// TIA Portal V18 export
DATA_BLOCK "ST10_Flow26_JMagnetLoad&Unload_iDB"   // DB1096
VERSION : 0.1
// stored: AutoNumber false, DBAccessibleFromOPCUA true, DBAccessibleFromWebserver true, InstanceOfName ST10_Flow26_JMagnetLoad&Unload, InstanceOfType FB
"ST10_Flow26_JMagnetLoad&Unload"
   // // inherited from GRAPH_BASE
   // VAR
   //    OFF_SQ_BASE : Bool;
   // END_VAR
   // VAR_INPUT
   //    iSysInface : "RCS_SysComInterface_V1";
   // END_VAR
   // VAR_IN_OUT
   //    ioPM_Inface : "RCS_PMInterface_V1";
   //    ioStatus : Int;
   // END_VAR
   // VAR
   //    sCtrlMode { S7_SetPoint := 'True'} : "SysFlowCtrlGraph";
   //    sUpdMES_Data : Bool;
   //    工件放行中 : Bool;
   //    前站站号 { ExternalAccessible := 'False'; ExternalVisible := 'False'; ExternalWritable := 'False'} : UInt;
   //    本站站号 { ExternalAccessible := 'False'; ExternalVisible := 'False'; ExternalWritable := 'False'} : UInt;
   //    弹窗Temp : Array[1..10] of Int;
   //    AlarmID : Int;
   //    TON { S7_SetPoint := 'True'} : Array[0..10] of TON_TIME;
   //    TOF { S7_SetPoint := 'True'} : Array[0..10] of TOF_TIME;
   //    sUP { S7_SetPoint := 'True'} : Array[0..10] of Bool;
   //    更新RFID完成 : Bool;
   //    RT_DATA { ExternalAccessible := 'False'; ExternalVisible := 'False'; ExternalWritable := 'False'; S7_SetPoint := 'True'} : G7_RTDataPlus_V6;
   //    Trans1 { ExternalAccessible := 'False'; ExternalVisible := 'False'; ExternalWritable := 'False'; S7_SetPoint := 'True'} : G7_TransitionPlus_V6;
   //    Trans2 { ExternalAccessible := 'False'; ExternalVisible := 'False'; ExternalWritable := 'False'; S7_SetPoint := 'True'} : G7_TransitionPlus_V6;
   //    Trans3 { ExternalAccessible := 'False'; ExternalVisible := 'False'; ExternalWritable := 'False'; S7_SetPoint := 'True'} : G7_TransitionPlus_V6;
   //    Trans102 { ExternalAccessible := 'False'; ExternalVisible := 'False'; ExternalWritable := 'False'; S7_SetPoint := 'True'} : G7_TransitionPlus_V6;
   //    Trans28 { ExternalAccessible := 'False'; ExternalVisible := 'False'; ExternalWritable := 'False'; S7_SetPoint := 'True'} : G7_TransitionPlus_V6;
   //    Trans29 { ExternalAccessible := 'False'; ExternalVisible := 'False'; ExternalWritable := 'False'; S7_SetPoint := 'True'} : G7_TransitionPlus_V6;
   //    Trans30 { ExternalAccessible := 'False'; ExternalVisible := 'False'; ExternalWritable := 'False'; S7_SetPoint := 'True'} : G7_TransitionPlus_V6;
   //    Trans31 { ExternalAccessible := 'False'; ExternalVisible := 'False'; ExternalWritable := 'False'; S7_SetPoint := 'True'} : G7_TransitionPlus_V6;
   //    Trans32 { ExternalAccessible := 'False'; ExternalVisible := 'False'; ExternalWritable := 'False'; S7_SetPoint := 'True'} : G7_TransitionPlus_V6;
   //    Trans33 { ExternalAccessible := 'False'; ExternalVisible := 'False'; ExternalWritable := 'False'; S7_SetPoint := 'True'} : G7_TransitionPlus_V6;
   //    Trans34 { ExternalAccessible := 'False'; ExternalVisible := 'False'; ExternalWritable := 'False'; S7_SetPoint := 'True'} : G7_TransitionPlus_V6;
   //    Trans35 { ExternalAccessible := 'False'; ExternalVisible := 'False'; ExternalWritable := 'False'; S7_SetPoint := 'True'} : G7_TransitionPlus_V6;
   //    Trans36 { ExternalAccessible := 'False'; ExternalVisible := 'False'; ExternalWritable := 'False'; S7_SetPoint := 'True'} : G7_TransitionPlus_V6;
   //    Trans37 { ExternalAccessible := 'False'; ExternalVisible := 'False'; ExternalWritable := 'False'; S7_SetPoint := 'True'} : G7_TransitionPlus_V6;
   //    Trans38 { ExternalAccessible := 'False'; ExternalVisible := 'False'; ExternalWritable := 'False'; S7_SetPoint := 'True'} : G7_TransitionPlus_V6;
   //    Trans39 { ExternalAccessible := 'False'; ExternalVisible := 'False'; ExternalWritable := 'False'; S7_SetPoint := 'True'} : G7_TransitionPlus_V6;
   //    Trans40 { ExternalAccessible := 'False'; ExternalVisible := 'False'; ExternalWritable := 'False'; S7_SetPoint := 'True'} : G7_TransitionPlus_V6;
   //    Trans41 { ExternalAccessible := 'False'; ExternalVisible := 'False'; ExternalWritable := 'False'; S7_SetPoint := 'True'} : G7_TransitionPlus_V6;
   //    Trans42 { ExternalAccessible := 'False'; ExternalVisible := 'False'; ExternalWritable := 'False'; S7_SetPoint := 'True'} : G7_TransitionPlus_V6;
   //    Trans43 { ExternalAccessible := 'False'; ExternalVisible := 'False'; ExternalWritable := 'False'; S7_SetPoint := 'True'} : G7_TransitionPlus_V6;
   //    Trans44 { ExternalAccessible := 'False'; ExternalVisible := 'False'; ExternalWritable := 'False'; S7_SetPoint := 'True'} : G7_TransitionPlus_V6;
   //    Trans45 { ExternalAccessible := 'False'; ExternalVisible := 'False'; ExternalWritable := 'False'; S7_SetPoint := 'True'} : G7_TransitionPlus_V6;
   //    Trans46 { ExternalAccessible := 'False'; ExternalVisible := 'False'; ExternalWritable := 'False'; S7_SetPoint := 'True'} : G7_TransitionPlus_V6;
   //    Trans47 { ExternalAccessible := 'False'; ExternalVisible := 'False'; ExternalWritable := 'False'; S7_SetPoint := 'True'} : G7_TransitionPlus_V6;
   //    Trans48 { ExternalAccessible := 'False'; ExternalVisible := 'False'; ExternalWritable := 'False'; S7_SetPoint := 'True'} : G7_TransitionPlus_V6;
   //    Trans49 { ExternalAccessible := 'False'; ExternalVisible := 'False'; ExternalWritable := 'False'; S7_SetPoint := 'True'} : G7_TransitionPlus_V6;
   //    Trans50 { ExternalAccessible := 'False'; ExternalVisible := 'False'; ExternalWritable := 'False'; S7_SetPoint := 'True'} : G7_TransitionPlus_V6;
   //    Trans51 { ExternalAccessible := 'False'; ExternalVisible := 'False'; ExternalWritable := 'False'; S7_SetPoint := 'True'} : G7_TransitionPlus_V6;
   //    Trans52 { ExternalAccessible := 'False'; ExternalVisible := 'False'; ExternalWritable := 'False'; S7_SetPoint := 'True'} : G7_TransitionPlus_V6;
   //    Trans53 { ExternalAccessible := 'False'; ExternalVisible := 'False'; ExternalWritable := 'False'; S7_SetPoint := 'True'} : G7_TransitionPlus_V6;
   //    Trans54 { ExternalAccessible := 'False'; ExternalVisible := 'False'; ExternalWritable := 'False'; S7_SetPoint := 'True'} : G7_TransitionPlus_V6;
   //    Trans55 { ExternalAccessible := 'False'; ExternalVisible := 'False'; ExternalWritable := 'False'; S7_SetPoint := 'True'} : G7_TransitionPlus_V6;
   //    Trans56 { ExternalAccessible := 'False'; ExternalVisible := 'False'; ExternalWritable := 'False'; S7_SetPoint := 'True'} : G7_TransitionPlus_V6;
   //    Trans57 { ExternalAccessible := 'False'; ExternalVisible := 'False'; ExternalWritable := 'False'; S7_SetPoint := 'True'} : G7_TransitionPlus_V6;
   //    Trans58 { ExternalAccessible := 'False'; ExternalVisible := 'False'; ExternalWritable := 'False'; S7_SetPoint := 'True'} : G7_TransitionPlus_V6;
   //    Trans59 { ExternalAccessible := 'False'; ExternalVisible := 'False'; ExternalWritable := 'False'; S7_SetPoint := 'True'} : G7_TransitionPlus_V6;
   //    Trans60 { ExternalAccessible := 'False'; ExternalVisible := 'False'; ExternalWritable := 'False'; S7_SetPoint := 'True'} : G7_TransitionPlus_V6;
   //    Trans61 { ExternalAccessible := 'False'; ExternalVisible := 'False'; ExternalWritable := 'False'; S7_SetPoint := 'True'} : G7_TransitionPlus_V6;
   //    Trans62 { ExternalAccessible := 'False'; ExternalVisible := 'False'; ExternalWritable := 'False'; S7_SetPoint := 'True'} : G7_TransitionPlus_V6;
   //    Trans63 { ExternalAccessible := 'False'; ExternalVisible := 'False'; ExternalWritable := 'False'; S7_SetPoint := 'True'} : G7_TransitionPlus_V6;
   //    Trans64 { ExternalAccessible := 'False'; ExternalVisible := 'False'; ExternalWritable := 'False'; S7_SetPoint := 'True'} : G7_TransitionPlus_V6;
   //    Trans65 { ExternalAccessible := 'False'; ExternalVisible := 'False'; ExternalWritable := 'False'; S7_SetPoint := 'True'} : G7_TransitionPlus_V6;
   //    Trans66 { ExternalAccessible := 'False'; ExternalVisible := 'False'; ExternalWritable := 'False'; S7_SetPoint := 'True'} : G7_TransitionPlus_V6;
   //    Trans67 { ExternalAccessible := 'False'; ExternalVisible := 'False'; ExternalWritable := 'False'; S7_SetPoint := 'True'} : G7_TransitionPlus_V6;
   //    Trans68 { ExternalAccessible := 'False'; ExternalVisible := 'False'; ExternalWritable := 'False'; S7_SetPoint := 'True'} : G7_TransitionPlus_V6;
   //    Trans69 { ExternalAccessible := 'False'; ExternalVisible := 'False'; ExternalWritable := 'False'; S7_SetPoint := 'True'} : G7_TransitionPlus_V6;
   //    Trans70 { ExternalAccessible := 'False'; ExternalVisible := 'False'; ExternalWritable := 'False'; S7_SetPoint := 'True'} : G7_TransitionPlus_V6;
   //    Trans71 { ExternalAccessible := 'False'; ExternalVisible := 'False'; ExternalWritable := 'False'; S7_SetPoint := 'True'} : G7_TransitionPlus_V6;
   //    Trans72 { ExternalAccessible := 'False'; ExternalVisible := 'False'; ExternalWritable := 'False'; S7_SetPoint := 'True'} : G7_TransitionPlus_V6;
   //    Trans73 { ExternalAccessible := 'False'; ExternalVisible := 'False'; ExternalWritable := 'False'; S7_SetPoint := 'True'} : G7_TransitionPlus_V6;
   //    Trans74 { ExternalAccessible := 'False'; ExternalVisible := 'False'; ExternalWritable := 'False'; S7_SetPoint := 'True'} : G7_TransitionPlus_V6;
   //    Trans75 { ExternalAccessible := 'False'; ExternalVisible := 'False'; ExternalWritable := 'False'; S7_SetPoint := 'True'} : G7_TransitionPlus_V6;
   //    Trans76 { ExternalAccessible := 'False'; ExternalVisible := 'False'; ExternalWritable := 'False'; S7_SetPoint := 'True'} : G7_TransitionPlus_V6;
   //    Trans77 { ExternalAccessible := 'False'; ExternalVisible := 'False'; ExternalWritable := 'False'; S7_SetPoint := 'True'} : G7_TransitionPlus_V6;
   //    Trans78 { ExternalAccessible := 'False'; ExternalVisible := 'False'; ExternalWritable := 'False'; S7_SetPoint := 'True'} : G7_TransitionPlus_V6;
   //    Trans79 { ExternalAccessible := 'False'; ExternalVisible := 'False'; ExternalWritable := 'False'; S7_SetPoint := 'True'} : G7_TransitionPlus_V6;
   //    Trans80 { ExternalAccessible := 'False'; ExternalVisible := 'False'; ExternalWritable := 'False'; S7_SetPoint := 'True'} : G7_TransitionPlus_V6;
   //    Trans81 { ExternalAccessible := 'False'; ExternalVisible := 'False'; ExternalWritable := 'False'; S7_SetPoint := 'True'} : G7_TransitionPlus_V6;
   //    Trans82 { ExternalAccessible := 'False'; ExternalVisible := 'False'; ExternalWritable := 'False'; S7_SetPoint := 'True'} : G7_TransitionPlus_V6;
   //    Trans200 { ExternalAccessible := 'False'; ExternalVisible := 'False'; ExternalWritable := 'False'; S7_SetPoint := 'True'} : G7_TransitionPlus_V6;
   //    Trans765 { ExternalAccessible := 'False'; ExternalVisible := 'False'; ExternalWritable := 'False'; S7_SetPoint := 'True'} : G7_TransitionPlus_V6;
   //    Trans766 { ExternalAccessible := 'False'; ExternalVisible := 'False'; ExternalWritable := 'False'; S7_SetPoint := 'True'} : G7_TransitionPlus_V6;
   //    Trans767 { ExternalAccessible := 'False'; ExternalVisible := 'False'; ExternalWritable := 'False'; S7_SetPoint := 'True'} : G7_TransitionPlus_V6;
   //    Trans119 { ExternalAccessible := 'False'; ExternalVisible := 'False'; ExternalWritable := 'False'; S7_SetPoint := 'True'} : G7_TransitionPlus_V6;
   //    Trans120 { ExternalAccessible := 'False'; ExternalVisible := 'False'; ExternalWritable := 'False'; S7_SetPoint := 'True'} : G7_TransitionPlus_V6;
   //    Trans121 { ExternalAccessible := 'False'; ExternalVisible := 'False'; ExternalWritable := 'False'; S7_SetPoint := 'True'} : G7_TransitionPlus_V6;
   //    Trans122 { ExternalAccessible := 'False'; ExternalVisible := 'False'; ExternalWritable := 'False'; S7_SetPoint := 'True'} : G7_TransitionPlus_V6;
   //    Trans123 { ExternalAccessible := 'False'; ExternalVisible := 'False'; ExternalWritable := 'False'; S7_SetPoint := 'True'} : G7_TransitionPlus_V6;
   //    Trans768 { ExternalAccessible := 'False'; ExternalVisible := 'False'; ExternalWritable := 'False'; S7_SetPoint := 'True'} : G7_TransitionPlus_V6;
   //    Trans769 { ExternalAccessible := 'False'; ExternalVisible := 'False'; ExternalWritable := 'False'; S7_SetPoint := 'True'} : G7_TransitionPlus_V6;
   //    Trans126 { ExternalAccessible := 'False'; ExternalVisible := 'False'; ExternalWritable := 'False'; S7_SetPoint := 'True'} : G7_TransitionPlus_V6;
   //    Trans127 { ExternalAccessible := 'False'; ExternalVisible := 'False'; ExternalWritable := 'False'; S7_SetPoint := 'True'} : G7_TransitionPlus_V6;
   //    Trans128 { ExternalAccessible := 'False'; ExternalVisible := 'False'; ExternalWritable := 'False'; S7_SetPoint := 'True'} : G7_TransitionPlus_V6;
   //    Trans124 { ExternalAccessible := 'False'; ExternalVisible := 'False'; ExternalWritable := 'False'; S7_SetPoint := 'True'} : G7_TransitionPlus_V6;
   //    Trans770 { ExternalAccessible := 'False'; ExternalVisible := 'False'; ExternalWritable := 'False'; S7_SetPoint := 'True'} : G7_TransitionPlus_V6;
   //    Trans771 { ExternalAccessible := 'False'; ExternalVisible := 'False'; ExternalWritable := 'False'; S7_SetPoint := 'True'} : G7_TransitionPlus_V6;
   //    Trans129 { ExternalAccessible := 'False'; ExternalVisible := 'False'; ExternalWritable := 'False'; S7_SetPoint := 'True'} : G7_TransitionPlus_V6;
   //    Trans130 { ExternalAccessible := 'False'; ExternalVisible := 'False'; ExternalWritable := 'False'; S7_SetPoint := 'True'} : G7_TransitionPlus_V6;
   //    Trans131 { ExternalAccessible := 'False'; ExternalVisible := 'False'; ExternalWritable := 'False'; S7_SetPoint := 'True'} : G7_TransitionPlus_V6;
   //    Trans125 { ExternalAccessible := 'False'; ExternalVisible := 'False'; ExternalWritable := 'False'; S7_SetPoint := 'True'} : G7_TransitionPlus_V6;
   //    Trans132 { ExternalAccessible := 'False'; ExternalVisible := 'False'; ExternalWritable := 'False'; S7_SetPoint := 'True'} : G7_TransitionPlus_V6;
   //    Trans772 { ExternalAccessible := 'False'; ExternalVisible := 'False'; ExternalWritable := 'False'; S7_SetPoint := 'True'} : G7_TransitionPlus_V6;
   //    Trans773 { ExternalAccessible := 'False'; ExternalVisible := 'False'; ExternalWritable := 'False'; S7_SetPoint := 'True'} : G7_TransitionPlus_V6;
   //    Trans133 { ExternalAccessible := 'False'; ExternalVisible := 'False'; ExternalWritable := 'False'; S7_SetPoint := 'True'} : G7_TransitionPlus_V6;
   //    Trans134 { ExternalAccessible := 'False'; ExternalVisible := 'False'; ExternalWritable := 'False'; S7_SetPoint := 'True'} : G7_TransitionPlus_V6;
   //    Trans776 { ExternalAccessible := 'False'; ExternalVisible := 'False'; ExternalWritable := 'False'; S7_SetPoint := 'True'} : G7_TransitionPlus_V6;
   //    Trans142 { ExternalAccessible := 'False'; ExternalVisible := 'False'; ExternalWritable := 'False'; S7_SetPoint := 'True'} : G7_TransitionPlus_V6;
   //    Trans143 { ExternalAccessible := 'False'; ExternalVisible := 'False'; ExternalWritable := 'False'; S7_SetPoint := 'True'} : G7_TransitionPlus_V6;
   //    Trans135 { ExternalAccessible := 'False'; ExternalVisible := 'False'; ExternalWritable := 'False'; S7_SetPoint := 'True'} : G7_TransitionPlus_V6;
   //    Trans136 { ExternalAccessible := 'False'; ExternalVisible := 'False'; ExternalWritable := 'False'; S7_SetPoint := 'True'} : G7_TransitionPlus_V6;
   //    Trans774 { ExternalAccessible := 'False'; ExternalVisible := 'False'; ExternalWritable := 'False'; S7_SetPoint := 'True'} : G7_TransitionPlus_V6;
   //    Trans775 { ExternalAccessible := 'False'; ExternalVisible := 'False'; ExternalWritable := 'False'; S7_SetPoint := 'True'} : G7_TransitionPlus_V6;
   //    Trans137 { ExternalAccessible := 'False'; ExternalVisible := 'False'; ExternalWritable := 'False'; S7_SetPoint := 'True'} : G7_TransitionPlus_V6;
   //    Trans138 { ExternalAccessible := 'False'; ExternalVisible := 'False'; ExternalWritable := 'False'; S7_SetPoint := 'True'} : G7_TransitionPlus_V6;
   //    Trans139 { ExternalAccessible := 'False'; ExternalVisible := 'False'; ExternalWritable := 'False'; S7_SetPoint := 'True'} : G7_TransitionPlus_V6;
   //    Trans140 { ExternalAccessible := 'False'; ExternalVisible := 'False'; ExternalWritable := 'False'; S7_SetPoint := 'True'} : G7_TransitionPlus_V6;
   //    Trans777 { ExternalAccessible := 'False'; ExternalVisible := 'False'; ExternalWritable := 'False'; S7_SetPoint := 'True'} : G7_TransitionPlus_V6;
   //    Trans778 { ExternalAccessible := 'False'; ExternalVisible := 'False'; ExternalWritable := 'False'; S7_SetPoint := 'True'} : G7_TransitionPlus_V6;
   //    Trans141 { ExternalAccessible := 'False'; ExternalVisible := 'False'; ExternalWritable := 'False'; S7_SetPoint := 'True'} : G7_TransitionPlus_V6;
   //    Trans144 { ExternalAccessible := 'False'; ExternalVisible := 'False'; ExternalWritable := 'False'; S7_SetPoint := 'True'} : G7_TransitionPlus_V6;
   //    Trans146 { ExternalAccessible := 'False'; ExternalVisible := 'False'; ExternalWritable := 'False'; S7_SetPoint := 'True'} : G7_TransitionPlus_V6;
   //    Trans147 { ExternalAccessible := 'False'; ExternalVisible := 'False'; ExternalWritable := 'False'; S7_SetPoint := 'True'} : G7_TransitionPlus_V6;
   //    Trans779 { ExternalAccessible := 'False'; ExternalVisible := 'False'; ExternalWritable := 'False'; S7_SetPoint := 'True'} : G7_TransitionPlus_V6;
   //    Trans780 { ExternalAccessible := 'False'; ExternalVisible := 'False'; ExternalWritable := 'False'; S7_SetPoint := 'True'} : G7_TransitionPlus_V6;
   //    Trans148 { ExternalAccessible := 'False'; ExternalVisible := 'False'; ExternalWritable := 'False'; S7_SetPoint := 'True'} : G7_TransitionPlus_V6;
   //    Trans149 { ExternalAccessible := 'False'; ExternalVisible := 'False'; ExternalWritable := 'False'; S7_SetPoint := 'True'} : G7_TransitionPlus_V6;
   //    Trans150 { ExternalAccessible := 'False'; ExternalVisible := 'False'; ExternalWritable := 'False'; S7_SetPoint := 'True'} : G7_TransitionPlus_V6;
   //    Trans163 { ExternalAccessible := 'False'; ExternalVisible := 'False'; ExternalWritable := 'False'; S7_SetPoint := 'True'} : G7_TransitionPlus_V6;
   //    Trans164 { ExternalAccessible := 'False'; ExternalVisible := 'False'; ExternalWritable := 'False'; S7_SetPoint := 'True'} : G7_TransitionPlus_V6;
   //    Trans165 { ExternalAccessible := 'False'; ExternalVisible := 'False'; ExternalWritable := 'False'; S7_SetPoint := 'True'} : G7_TransitionPlus_V6;
   //    Trans166 { ExternalAccessible := 'False'; ExternalVisible := 'False'; ExternalWritable := 'False'; S7_SetPoint := 'True'} : G7_TransitionPlus_V6;
   //    Trans167 { ExternalAccessible := 'False'; ExternalVisible := 'False'; ExternalWritable := 'False'; S7_SetPoint := 'True'} : G7_TransitionPlus_V6;
   //    Trans151 { ExternalAccessible := 'False'; ExternalVisible := 'False'; ExternalWritable := 'False'; S7_SetPoint := 'True'} : G7_TransitionPlus_V6;
   //    Trans152 { ExternalAccessible := 'False'; ExternalVisible := 'False'; ExternalWritable := 'False'; S7_SetPoint := 'True'} : G7_TransitionPlus_V6;
   //    Trans153 { ExternalAccessible := 'False'; ExternalVisible := 'False'; ExternalWritable := 'False'; S7_SetPoint := 'True'} : G7_TransitionPlus_V6;
   //    Trans168 { ExternalAccessible := 'False'; ExternalVisible := 'False'; ExternalWritable := 'False'; S7_SetPoint := 'True'} : G7_TransitionPlus_V6;
   //    Trans781 { ExternalAccessible := 'False'; ExternalVisible := 'False'; ExternalWritable := 'False'; S7_SetPoint := 'True'} : G7_TransitionPlus_V6;
   //    Trans782 { ExternalAccessible := 'False'; ExternalVisible := 'False'; ExternalWritable := 'False'; S7_SetPoint := 'True'} : G7_TransitionPlus_V6;
   //    Trans783 { ExternalAccessible := 'False'; ExternalVisible := 'False'; ExternalWritable := 'False'; S7_SetPoint := 'True'} : G7_TransitionPlus_V6;
   //    Trans154 { ExternalAccessible := 'False'; ExternalVisible := 'False'; ExternalWritable := 'False'; S7_SetPoint := 'True'} : G7_TransitionPlus_V6;
   //    Trans155 { ExternalAccessible := 'False'; ExternalVisible := 'False'; ExternalWritable := 'False'; S7_SetPoint := 'True'} : G7_TransitionPlus_V6;
   //    Trans784 { ExternalAccessible := 'False'; ExternalVisible := 'False'; ExternalWritable := 'False'; S7_SetPoint := 'True'} : G7_TransitionPlus_V6;
   //    Trans785 { ExternalAccessible := 'False'; ExternalVisible := 'False'; ExternalWritable := 'False'; S7_SetPoint := 'True'} : G7_TransitionPlus_V6;
   //    Trans156 { ExternalAccessible := 'False'; ExternalVisible := 'False'; ExternalWritable := 'False'; S7_SetPoint := 'True'} : G7_TransitionPlus_V6;
   //    Trans157 { ExternalAccessible := 'False'; ExternalVisible := 'False'; ExternalWritable := 'False'; S7_SetPoint := 'True'} : G7_TransitionPlus_V6;
   //    Trans158 { ExternalAccessible := 'False'; ExternalVisible := 'False'; ExternalWritable := 'False'; S7_SetPoint := 'True'} : G7_TransitionPlus_V6;
   //    Trans159 { ExternalAccessible := 'False'; ExternalVisible := 'False'; ExternalWritable := 'False'; S7_SetPoint := 'True'} : G7_TransitionPlus_V6;
   //    Trans786 { ExternalAccessible := 'False'; ExternalVisible := 'False'; ExternalWritable := 'False'; S7_SetPoint := 'True'} : G7_TransitionPlus_V6;
   //    Trans787 { ExternalAccessible := 'False'; ExternalVisible := 'False'; ExternalWritable := 'False'; S7_SetPoint := 'True'} : G7_TransitionPlus_V6;
   //    Trans160 { ExternalAccessible := 'False'; ExternalVisible := 'False'; ExternalWritable := 'False'; S7_SetPoint := 'True'} : G7_TransitionPlus_V6;
   //    Trans161 { ExternalAccessible := 'False'; ExternalVisible := 'False'; ExternalWritable := 'False'; S7_SetPoint := 'True'} : G7_TransitionPlus_V6;
   //    Trans162 { ExternalAccessible := 'False'; ExternalVisible := 'False'; ExternalWritable := 'False'; S7_SetPoint := 'True'} : G7_TransitionPlus_V6;
   //    Trans169 { ExternalAccessible := 'False'; ExternalVisible := 'False'; ExternalWritable := 'False'; S7_SetPoint := 'True'} : G7_TransitionPlus_V6;
   //    Trans788 { ExternalAccessible := 'False'; ExternalVisible := 'False'; ExternalWritable := 'False'; S7_SetPoint := 'True'} : G7_TransitionPlus_V6;
   //    Trans789 { ExternalAccessible := 'False'; ExternalVisible := 'False'; ExternalWritable := 'False'; S7_SetPoint := 'True'} : G7_TransitionPlus_V6;
   //    Trans170 { ExternalAccessible := 'False'; ExternalVisible := 'False'; ExternalWritable := 'False'; S7_SetPoint := 'True'} : G7_TransitionPlus_V6;
   //    Trans171 { ExternalAccessible := 'False'; ExternalVisible := 'False'; ExternalWritable := 'False'; S7_SetPoint := 'True'} : G7_TransitionPlus_V6;
   //    Trans172 { ExternalAccessible := 'False'; ExternalVisible := 'False'; ExternalWritable := 'False'; S7_SetPoint := 'True'} : G7_TransitionPlus_V6;
   //    Trans173 { ExternalAccessible := 'False'; ExternalVisible := 'False'; ExternalWritable := 'False'; S7_SetPoint := 'True'} : G7_TransitionPlus_V6;
   //    Trans174 { ExternalAccessible := 'False'; ExternalVisible := 'False'; ExternalWritable := 'False'; S7_SetPoint := 'True'} : G7_TransitionPlus_V6;
   //    Trans175 { ExternalAccessible := 'False'; ExternalVisible := 'False'; ExternalWritable := 'False'; S7_SetPoint := 'True'} : G7_TransitionPlus_V6;
   //    Trans197 { ExternalAccessible := 'False'; ExternalVisible := 'False'; ExternalWritable := 'False'; S7_SetPoint := 'True'} : G7_TransitionPlus_V6;
   //    Trans198 { ExternalAccessible := 'False'; ExternalVisible := 'False'; ExternalWritable := 'False'; S7_SetPoint := 'True'} : G7_TransitionPlus_V6;
   //    Trans176 { ExternalAccessible := 'False'; ExternalVisible := 'False'; ExternalWritable := 'False'; S7_SetPoint := 'True'} : G7_TransitionPlus_V6;
   //    Trans145 { ExternalAccessible := 'False'; ExternalVisible := 'False'; ExternalWritable := 'False'; S7_SetPoint := 'True'} : G7_TransitionPlus_V6;
   //    Trans177 { ExternalAccessible := 'False'; ExternalVisible := 'False'; ExternalWritable := 'False'; S7_SetPoint := 'True'} : G7_TransitionPlus_V6;
   //    Trans202 { ExternalAccessible := 'False'; ExternalVisible := 'False'; ExternalWritable := 'False'; S7_SetPoint := 'True'} : G7_TransitionPlus_V6;
   //    Trans203 { ExternalAccessible := 'False'; ExternalVisible := 'False'; ExternalWritable := 'False'; S7_SetPoint := 'True'} : G7_TransitionPlus_V6;
   //    Trans204 { ExternalAccessible := 'False'; ExternalVisible := 'False'; ExternalWritable := 'False'; S7_SetPoint := 'True'} : G7_TransitionPlus_V6;
   //    Trans205 { ExternalAccessible := 'False'; ExternalVisible := 'False'; ExternalWritable := 'False'; S7_SetPoint := 'True'} : G7_TransitionPlus_V6;
   //    Trans206 { ExternalAccessible := 'False'; ExternalVisible := 'False'; ExternalWritable := 'False'; S7_SetPoint := 'True'} : G7_TransitionPlus_V6;
   //    Trans207 { ExternalAccessible := 'False'; ExternalVisible := 'False'; ExternalWritable := 'False'; S7_SetPoint := 'True'} : G7_TransitionPlus_V6;
   //    Trans250 { ExternalAccessible := 'False'; ExternalVisible := 'False'; ExternalWritable := 'False'; S7_SetPoint := 'True'} : G7_TransitionPlus_V6;
   //    Trans251 { ExternalAccessible := 'False'; ExternalVisible := 'False'; ExternalWritable := 'False'; S7_SetPoint := 'True'} : G7_TransitionPlus_V6;
   //    Trans252 { ExternalAccessible := 'False'; ExternalVisible := 'False'; ExternalWritable := 'False'; S7_SetPoint := 'True'} : G7_TransitionPlus_V6;
   //    Trans253 { ExternalAccessible := 'False'; ExternalVisible := 'False'; ExternalWritable := 'False'; S7_SetPoint := 'True'} : G7_TransitionPlus_V6;
   //    Trans254 { ExternalAccessible := 'False'; ExternalVisible := 'False'; ExternalWritable := 'False'; S7_SetPoint := 'True'} : G7_TransitionPlus_V6;
   //    Trans255 { ExternalAccessible := 'False'; ExternalVisible := 'False'; ExternalWritable := 'False'; S7_SetPoint := 'True'} : G7_TransitionPlus_V6;
   //    Trans256 { ExternalAccessible := 'False'; ExternalVisible := 'False'; ExternalWritable := 'False'; S7_SetPoint := 'True'} : G7_TransitionPlus_V6;
   //    Trans257 { ExternalAccessible := 'False'; ExternalVisible := 'False'; ExternalWritable := 'False'; S7_SetPoint := 'True'} : G7_TransitionPlus_V6;
   //    Trans258 { ExternalAccessible := 'False'; ExternalVisible := 'False'; ExternalWritable := 'False'; S7_SetPoint := 'True'} : G7_TransitionPlus_V6;
   //    Trans259 { ExternalAccessible := 'False'; ExternalVisible := 'False'; ExternalWritable := 'False'; S7_SetPoint := 'True'} : G7_TransitionPlus_V6;
   //    Trans260 { ExternalAccessible := 'False'; ExternalVisible := 'False'; ExternalWritable := 'False'; S7_SetPoint := 'True'} : G7_TransitionPlus_V6;
   //    Trans613 { ExternalAccessible := 'False'; ExternalVisible := 'False'; ExternalWritable := 'False'; S7_SetPoint := 'True'} : G7_TransitionPlus_V6;
   //    F26_Initial { ExternalAccessible := 'False'; ExternalVisible := 'False'; ExternalWritable := 'False'; S7_SetPoint := 'True'} : G7_StepPlus_V6;
   //    S2 { ExternalAccessible := 'False'; ExternalVisible := 'False'; ExternalWritable := 'False'; S7_SetPoint := 'True'} : G7_StepPlus_V6;
   //    S3 { ExternalAccessible := 'False'; ExternalVisible := 'False'; ExternalWritable := 'False'; S7_SetPoint := 'True'} : G7_StepPlus_V6;
   //    S4 { ExternalAccessible := 'False'; ExternalVisible := 'False'; ExternalWritable := 'False'; S7_SetPoint := 'True'} : G7_StepPlus_V6;
   //    S10_InitialFinish { ExternalAccessible := 'False'; ExternalVisible := 'False'; ExternalWritable := 'False'; S7_SetPoint := 'True'} : G7_StepPlus_V6;
   //    MotorCWStart { ExternalAccessible := 'False'; ExternalVisible := 'False'; ExternalWritable := 'False'; S7_SetPoint := 'True'} : G7_StepPlus_V6;
   //    MotorCWStart_1 { ExternalAccessible := 'False'; ExternalVisible := 'False'; ExternalWritable := 'False'; S7_SetPoint := 'True'} : G7_StepPlus_V6;
   //    MotorRunDelay { ExternalAccessible := 'False'; ExternalVisible := 'False'; ExternalWritable := 'False'; S7_SetPoint := 'True'} : G7_StepPlus_V6;
   //    MotorRunDelay_1 { ExternalAccessible := 'False'; ExternalVisible := 'False'; ExternalWritable := 'False'; S7_SetPoint := 'True'} : G7_StepPlus_V6;
   //    StopProcess { ExternalAccessible := 'False'; ExternalVisible := 'False'; ExternalWritable := 'False'; S7_SetPoint := 'True'} : G7_StepPlus_V6;
   //    LoadingStop_2 { ExternalAccessible := 'False'; ExternalVisible := 'False'; ExternalWritable := 'False'; S7_SetPoint := 'True'} : G7_StepPlus_V6;
   //    LoadingStop_3 { ExternalAccessible := 'False'; ExternalVisible := 'False'; ExternalWritable := 'False'; S7_SetPoint := 'True'} : G7_StepPlus_V6;
   //    LoadingStop_4 { ExternalAccessible := 'False'; ExternalVisible := 'False'; ExternalWritable := 'False'; S7_SetPoint := 'True'} : G7_StepPlus_V6;
   //    CheckPalletExist { ExternalAccessible := 'False'; ExternalVisible := 'False'; ExternalWritable := 'False'; S7_SetPoint := 'True'} : G7_StepPlus_V6;
   //    CheckPalletExist_1 { ExternalAccessible := 'False'; ExternalVisible := 'False'; ExternalWritable := 'False'; S7_SetPoint := 'True'} : G7_StepPlus_V6;
   //    CheckMaterialDoorLock { ExternalAccessible := 'False'; ExternalVisible := 'False'; ExternalWritable := 'False'; S7_SetPoint := 'True'} : G7_StepPlus_V6;
   //    MotorRun { ExternalAccessible := 'False'; ExternalVisible := 'False'; ExternalWritable := 'False'; S7_SetPoint := 'True'} : G7_StepPlus_V6;
   //    WaitLineMotorReady { ExternalAccessible := 'False'; ExternalVisible := 'False'; ExternalWritable := 'False'; S7_SetPoint := 'True'} : G7_StepPlus_V6;
   //    WaitPalletRequestRelease { ExternalAccessible := 'False'; ExternalVisible := 'False'; ExternalWritable := 'False'; S7_SetPoint := 'True'} : G7_StepPlus_V6;
   //    WaitPalletArrveNextPos { ExternalAccessible := 'False'; ExternalVisible := 'False'; ExternalWritable := 'False'; S7_SetPoint := 'True'} : G7_StepPlus_V6;
   //    WaitLineMotorReady_1 { ExternalAccessible := 'False'; ExternalVisible := 'False'; ExternalWritable := 'False'; S7_SetPoint := 'True'} : G7_StepPlus_V6;
   //    WaitPalletRequestRelease_1 { ExternalAccessible := 'False'; ExternalVisible := 'False'; ExternalWritable := 'False'; S7_SetPoint := 'True'} : G7_StepPlus_V6;
   //    WaitPalletArrveNextPos_1 { ExternalAccessible := 'False'; ExternalVisible := 'False'; ExternalWritable := 'False'; S7_SetPoint := 'True'} : G7_StepPlus_V6;
   //    CheckPalletExist_2 { ExternalAccessible := 'False'; ExternalVisible := 'False'; ExternalWritable := 'False'; S7_SetPoint := 'True'} : G7_StepPlus_V6;
   //    WaitLineMotorReady_2 { ExternalAccessible := 'False'; ExternalVisible := 'False'; ExternalWritable := 'False'; S7_SetPoint := 'True'} : G7_StepPlus_V6;
   //    WaitPalletRequestRelease_2 { ExternalAccessible := 'False'; ExternalVisible := 'False'; ExternalWritable := 'False'; S7_SetPoint := 'True'} : G7_StepPlus_V6;
   //    WaitPalletArrveNextPos_2 { ExternalAccessible := 'False'; ExternalVisible := 'False'; ExternalWritable := 'False'; S7_SetPoint := 'True'} : G7_StepPlus_V6;
   //    CheckPalletExist_3 { ExternalAccessible := 'False'; ExternalVisible := 'False'; ExternalWritable := 'False'; S7_SetPoint := 'True'} : G7_StepPlus_V6;
   //    WaitLineMotorReady_3 { ExternalAccessible := 'False'; ExternalVisible := 'False'; ExternalWritable := 'False'; S7_SetPoint := 'True'} : G7_StepPlus_V6;
   //    WaitPalletRequestRelease_3 { ExternalAccessible := 'False'; ExternalVisible := 'False'; ExternalWritable := 'False'; S7_SetPoint := 'True'} : G7_StepPlus_V6;
   //    WaitPalletArrveNextPos_3 { ExternalAccessible := 'False'; ExternalVisible := 'False'; ExternalWritable := 'False'; S7_SetPoint := 'True'} : G7_StepPlus_V6;
   //    CheckPalletExist_4 { ExternalAccessible := 'False'; ExternalVisible := 'False'; ExternalWritable := 'False'; S7_SetPoint := 'True'} : G7_StepPlus_V6;
   //    WaitLineMotorReady_4 { ExternalAccessible := 'False'; ExternalVisible := 'False'; ExternalWritable := 'False'; S7_SetPoint := 'True'} : G7_StepPlus_V6;
   //    WaitPalletRequestRelease_4 { ExternalAccessible := 'False'; ExternalVisible := 'False'; ExternalWritable := 'False'; S7_SetPoint := 'True'} : G7_StepPlus_V6;
   //    WaitPalletArrveNextPos_4 { ExternalAccessible := 'False'; ExternalVisible := 'False'; ExternalWritable := 'False'; S7_SetPoint := 'True'} : G7_StepPlus_V6;
   //    CheckPalletExist_5 { ExternalAccessible := 'False'; ExternalVisible := 'False'; ExternalWritable := 'False'; S7_SetPoint := 'True'} : G7_StepPlus_V6;
   //    WaitLineMotorReady_5 { ExternalAccessible := 'False'; ExternalVisible := 'False'; ExternalWritable := 'False'; S7_SetPoint := 'True'} : G7_StepPlus_V6;
   //    WaitPalletRequestRelease_5 { ExternalAccessible := 'False'; ExternalVisible := 'False'; ExternalWritable := 'False'; S7_SetPoint := 'True'} : G7_StepPlus_V6;
   //    WaitPalletArrveNextPos_5 { ExternalAccessible := 'False'; ExternalVisible := 'False'; ExternalWritable := 'False'; S7_SetPoint := 'True'} : G7_StepPlus_V6;
   //    CheckPalletExist_6 { ExternalAccessible := 'False'; ExternalVisible := 'False'; ExternalWritable := 'False'; S7_SetPoint := 'True'} : G7_StepPlus_V6;
   //    WaitLineMotorReady_6 { ExternalAccessible := 'False'; ExternalVisible := 'False'; ExternalWritable := 'False'; S7_SetPoint := 'True'} : G7_StepPlus_V6;
   //    WaitPalletRequestRelease_6 { ExternalAccessible := 'False'; ExternalVisible := 'False'; ExternalWritable := 'False'; S7_SetPoint := 'True'} : G7_StepPlus_V6;
   //    WaitPalletArrveNextPos_6 { ExternalAccessible := 'False'; ExternalVisible := 'False'; ExternalWritable := 'False'; S7_SetPoint := 'True'} : G7_StepPlus_V6;
   //    LoadStop_14 { ExternalAccessible := 'False'; ExternalVisible := 'False'; ExternalWritable := 'False'; S7_SetPoint := 'True'} : G7_StepPlus_V6;
   //    LoadStop_12 { ExternalAccessible := 'False'; ExternalVisible := 'False'; ExternalWritable := 'False'; S7_SetPoint := 'True'} : G7_StepPlus_V6;
   //    LoadStop_13 { ExternalAccessible := 'False'; ExternalVisible := 'False'; ExternalWritable := 'False'; S7_SetPoint := 'True'} : G7_StepPlus_V6;
   //    CheckPalletExist_7 { ExternalAccessible := 'False'; ExternalVisible := 'False'; ExternalWritable := 'False'; S7_SetPoint := 'True'} : G7_StepPlus_V6;
   //    WaitLineMotorReady_7 { ExternalAccessible := 'False'; ExternalVisible := 'False'; ExternalWritable := 'False'; S7_SetPoint := 'True'} : G7_StepPlus_V6;
   //    WaitPalletRequestRelease_7 { ExternalAccessible := 'False'; ExternalVisible := 'False'; ExternalWritable := 'False'; S7_SetPoint := 'True'} : G7_StepPlus_V6;
   //    WaitPalletArrveNextPos_7 { ExternalAccessible := 'False'; ExternalVisible := 'False'; ExternalWritable := 'False'; S7_SetPoint := 'True'} : G7_StepPlus_V6;
   //    CheckPalletExist_8 { ExternalAccessible := 'False'; ExternalVisible := 'False'; ExternalWritable := 'False'; S7_SetPoint := 'True'} : G7_StepPlus_V6;
   //    WaitLineMotorReady_8 { ExternalAccessible := 'False'; ExternalVisible := 'False'; ExternalWritable := 'False'; S7_SetPoint := 'True'} : G7_StepPlus_V6;
   //    WaitPalletRequestRelease_8 { ExternalAccessible := 'False'; ExternalVisible := 'False'; ExternalWritable := 'False'; S7_SetPoint := 'True'} : G7_StepPlus_V6;
   //    WaitPalletArrveNextPos_8 { ExternalAccessible := 'False'; ExternalVisible := 'False'; ExternalWritable := 'False'; S7_SetPoint := 'True'} : G7_StepPlus_V6;
   //    CheckPalletExist_9 { ExternalAccessible := 'False'; ExternalVisible := 'False'; ExternalWritable := 'False'; S7_SetPoint := 'True'} : G7_StepPlus_V6;
   //    WaitLineMotorReady_9 { ExternalAccessible := 'False'; ExternalVisible := 'False'; ExternalWritable := 'False'; S7_SetPoint := 'True'} : G7_StepPlus_V6;
   //    WaitPalletRequestRelease_9 { ExternalAccessible := 'False'; ExternalVisible := 'False'; ExternalWritable := 'False'; S7_SetPoint := 'True'} : G7_StepPlus_V6;
   //    WaitPalletArrveNextPos_9 { ExternalAccessible := 'False'; ExternalVisible := 'False'; ExternalWritable := 'False'; S7_SetPoint := 'True'} : G7_StepPlus_V6;
   //    CheckPalletExist_10 { ExternalAccessible := 'False'; ExternalVisible := 'False'; ExternalWritable := 'False'; S7_SetPoint := 'True'} : G7_StepPlus_V6;
   //    WaitLineMotorReady_10 { ExternalAccessible := 'False'; ExternalVisible := 'False'; ExternalWritable := 'False'; S7_SetPoint := 'True'} : G7_StepPlus_V6;
   //    WaitPalletRequestRelease_10 { ExternalAccessible := 'False'; ExternalVisible := 'False'; ExternalWritable := 'False'; S7_SetPoint := 'True'} : G7_StepPlus_V6;
   //    WaitPalletArrveNextPos_10 { ExternalAccessible := 'False'; ExternalVisible := 'False'; ExternalWritable := 'False'; S7_SetPoint := 'True'} : G7_StepPlus_V6;
   //    MotorRun_1 { ExternalAccessible := 'False'; ExternalVisible := 'False'; ExternalWritable := 'False'; S7_SetPoint := 'True'} : G7_StepPlus_V6;
   //    "MiddleNoPallet?" { ExternalAccessible := 'False'; ExternalVisible := 'False'; ExternalWritable := 'False'; S7_SetPoint := 'True'} : G7_StepPlus_V6;
   //    ProcessStart { ExternalAccessible := 'False'; ExternalVisible := 'False'; ExternalWritable := 'False'; S7_SetPoint := 'True'} : G7_StepPlus_V6;
   //    StoperReset { ExternalAccessible := 'False'; ExternalVisible := 'False'; ExternalWritable := 'False'; S7_SetPoint := 'True'} : G7_StepPlus_V6;
   //    StoperReset_1 { ExternalAccessible := 'False'; ExternalVisible := 'False'; ExternalWritable := 'False'; S7_SetPoint := 'True'} : G7_StepPlus_V6;
   //    StoperRelease_1 { ExternalAccessible := 'False'; ExternalVisible := 'False'; ExternalWritable := 'False'; S7_SetPoint := 'True'} : G7_StepPlus_V6;
   //    AriveTimeDelay_1 { ExternalAccessible := 'False'; ExternalVisible := 'False'; ExternalWritable := 'False'; S7_SetPoint := 'True'} : G7_StepPlus_V6;
   //    AriveTimeDelay_2 { ExternalAccessible := 'False'; ExternalVisible := 'False'; ExternalWritable := 'False'; S7_SetPoint := 'True'} : G7_StepPlus_V6;
   //    StoperReset_2 { ExternalAccessible := 'False'; ExternalVisible := 'False'; ExternalWritable := 'False'; S7_SetPoint := 'True'} : G7_StepPlus_V6;
   //    StoperRelease_2 { ExternalAccessible := 'False'; ExternalVisible := 'False'; ExternalWritable := 'False'; S7_SetPoint := 'True'} : G7_StepPlus_V6;
   //    WaitPalletArive { ExternalAccessible := 'False'; ExternalVisible := 'False'; ExternalWritable := 'False'; S7_SetPoint := 'True'} : G7_StepPlus_V6;
   //    TimeDelay { ExternalAccessible := 'False'; ExternalVisible := 'False'; ExternalWritable := 'False'; S7_SetPoint := 'True'} : G7_StepPlus_V6;
   //    AriveTimeDelay_3 { ExternalAccessible := 'False'; ExternalVisible := 'False'; ExternalWritable := 'False'; S7_SetPoint := 'True'} : G7_StepPlus_V6;
   //    StoperReset_3 { ExternalAccessible := 'False'; ExternalVisible := 'False'; ExternalWritable := 'False'; S7_SetPoint := 'True'} : G7_StepPlus_V6;
   //    StoperRelease_3 { ExternalAccessible := 'False'; ExternalVisible := 'False'; ExternalWritable := 'False'; S7_SetPoint := 'True'} : G7_StepPlus_V6;
   //    WaitPalletArive_1 { ExternalAccessible := 'False'; ExternalVisible := 'False'; ExternalWritable := 'False'; S7_SetPoint := 'True'} : G7_StepPlus_V6;
   //    TimeDelay_1 { ExternalAccessible := 'False'; ExternalVisible := 'False'; ExternalWritable := 'False'; S7_SetPoint := 'True'} : G7_StepPlus_V6;
   //    AriveTimeDelay_4 { ExternalAccessible := 'False'; ExternalVisible := 'False'; ExternalWritable := 'False'; S7_SetPoint := 'True'} : G7_StepPlus_V6;
   //    StoperReset_4 { ExternalAccessible := 'False'; ExternalVisible := 'False'; ExternalWritable := 'False'; S7_SetPoint := 'True'} : G7_StepPlus_V6;
   //    MotorStop { ExternalAccessible := 'False'; ExternalVisible := 'False'; ExternalWritable := 'False'; S7_SetPoint := 'True'} : G7_StepPlus_V6;
   //    StoperRelease_4 { ExternalAccessible := 'False'; ExternalVisible := 'False'; ExternalWritable := 'False'; S7_SetPoint := 'True'} : G7_StepPlus_V6;
   //    WaitPalletArive_2 { ExternalAccessible := 'False'; ExternalVisible := 'False'; ExternalWritable := 'False'; S7_SetPoint := 'True'} : G7_StepPlus_V6;
   //    TimeDelay_2 { ExternalAccessible := 'False'; ExternalVisible := 'False'; ExternalWritable := 'False'; S7_SetPoint := 'True'} : G7_StepPlus_V6;
   //    AriveTimeDelay_5 { ExternalAccessible := 'False'; ExternalVisible := 'False'; ExternalWritable := 'False'; S7_SetPoint := 'True'} : G7_StepPlus_V6;
   //    StoperReset_5 { ExternalAccessible := 'False'; ExternalVisible := 'False'; ExternalWritable := 'False'; S7_SetPoint := 'True'} : G7_StepPlus_V6;
   //    StoperRelease_5 { ExternalAccessible := 'False'; ExternalVisible := 'False'; ExternalWritable := 'False'; S7_SetPoint := 'True'} : G7_StepPlus_V6;
   //    WaitPalletArive_3 { ExternalAccessible := 'False'; ExternalVisible := 'False'; ExternalWritable := 'False'; S7_SetPoint := 'True'} : G7_StepPlus_V6;
   //    TimeDelay_3 { ExternalAccessible := 'False'; ExternalVisible := 'False'; ExternalWritable := 'False'; S7_SetPoint := 'True'} : G7_StepPlus_V6;
   //    AriveTimeDelay_6 { ExternalAccessible := 'False'; ExternalVisible := 'False'; ExternalWritable := 'False'; S7_SetPoint := 'True'} : G7_StepPlus_V6;
   //    LoadingStop_1 { ExternalAccessible := 'False'; ExternalVisible := 'False'; ExternalWritable := 'False'; S7_SetPoint := 'True'} : G7_StepPlus_V6;
   //    Step143 { ExternalAccessible := 'False'; ExternalVisible := 'False'; ExternalWritable := 'False'; S7_SetPoint := 'True'} : G7_StepPlus_V6;
   //    StoperReset_6 { ExternalAccessible := 'False'; ExternalVisible := 'False'; ExternalWritable := 'False'; S7_SetPoint := 'True'} : G7_StepPlus_V6;
   //    StoperRelease_6 { ExternalAccessible := 'False'; ExternalVisible := 'False'; ExternalWritable := 'False'; S7_SetPoint := 'True'} : G7_StepPlus_V6;
   //    WaitPalletArive_4 { ExternalAccessible := 'False'; ExternalVisible := 'False'; ExternalWritable := 'False'; S7_SetPoint := 'True'} : G7_StepPlus_V6;
   //    TimeDelay_4 { ExternalAccessible := 'False'; ExternalVisible := 'False'; ExternalWritable := 'False'; S7_SetPoint := 'True'} : G7_StepPlus_V6;
   //    AriveTimeDelay_7 { ExternalAccessible := 'False'; ExternalVisible := 'False'; ExternalWritable := 'False'; S7_SetPoint := 'True'} : G7_StepPlus_V6;
   //    StoperReset_7 { ExternalAccessible := 'False'; ExternalVisible := 'False'; ExternalWritable := 'False'; S7_SetPoint := 'True'} : G7_StepPlus_V6;
   //    StoperRelease_7 { ExternalAccessible := 'False'; ExternalVisible := 'False'; ExternalWritable := 'False'; S7_SetPoint := 'True'} : G7_StepPlus_V6;
   //    WaitPalletArive_5 { ExternalAccessible := 'False'; ExternalVisible := 'False'; ExternalWritable := 'False'; S7_SetPoint := 'True'} : G7_StepPlus_V6;
   //    TimeDelay_5 { ExternalAccessible := 'False'; ExternalVisible := 'False'; ExternalWritable := 'False'; S7_SetPoint := 'True'} : G7_StepPlus_V6;
   //    Step153 { ExternalAccessible := 'False'; ExternalVisible := 'False'; ExternalWritable := 'False'; S7_SetPoint := 'True'} : G7_StepPlus_V6;
   //    "CheckMachine Mode_1" { ExternalAccessible := 'False'; ExternalVisible := 'False'; ExternalWritable := 'False'; S7_SetPoint := 'True'} : G7_StepPlus_V6;
   //    "CheckMachine Mode_2" { ExternalAccessible := 'False'; ExternalVisible := 'False'; ExternalWritable := 'False'; S7_SetPoint := 'True'} : G7_StepPlus_V6;
   //    "CheckMachine Mode_3" { ExternalAccessible := 'False'; ExternalVisible := 'False'; ExternalWritable := 'False'; S7_SetPoint := 'True'} : G7_StepPlus_V6;
   //    "CheckMachine Mode_4" { ExternalAccessible := 'False'; ExternalVisible := 'False'; ExternalWritable := 'False'; S7_SetPoint := 'True'} : G7_StepPlus_V6;
   //    "CheckMachine Mode_5" { ExternalAccessible := 'False'; ExternalVisible := 'False'; ExternalWritable := 'False'; S7_SetPoint := 'True'} : G7_StepPlus_V6;
   //    AriveTimeDelay_8 { ExternalAccessible := 'False'; ExternalVisible := 'False'; ExternalWritable := 'False'; S7_SetPoint := 'True'} : G7_StepPlus_V6;
   //    LoadStop_11 { ExternalAccessible := 'False'; ExternalVisible := 'False'; ExternalWritable := 'False'; S7_SetPoint := 'True'} : G7_StepPlus_V6;
   //    StoperReset_8 { ExternalAccessible := 'False'; ExternalVisible := 'False'; ExternalWritable := 'False'; S7_SetPoint := 'True'} : G7_StepPlus_V6;
   //    StoperRelease_8 { ExternalAccessible := 'False'; ExternalVisible := 'False'; ExternalWritable := 'False'; S7_SetPoint := 'True'} : G7_StepPlus_V6;
   //    AriveTimeDelay_9 { ExternalAccessible := 'False'; ExternalVisible := 'False'; ExternalWritable := 'False'; S7_SetPoint := 'True'} : G7_StepPlus_V6;
   //    StoperReset_9 { ExternalAccessible := 'False'; ExternalVisible := 'False'; ExternalWritable := 'False'; S7_SetPoint := 'True'} : G7_StepPlus_V6;
   //    StoperRelease_9 { ExternalAccessible := 'False'; ExternalVisible := 'False'; ExternalWritable := 'False'; S7_SetPoint := 'True'} : G7_StepPlus_V6;
   //    WaitPalletArive_6 { ExternalAccessible := 'False'; ExternalVisible := 'False'; ExternalWritable := 'False'; S7_SetPoint := 'True'} : G7_StepPlus_V6;
   //    TimeDelay_6 { ExternalAccessible := 'False'; ExternalVisible := 'False'; ExternalWritable := 'False'; S7_SetPoint := 'True'} : G7_StepPlus_V6;
   //    AriveTimeDelay_10 { ExternalAccessible := 'False'; ExternalVisible := 'False'; ExternalWritable := 'False'; S7_SetPoint := 'True'} : G7_StepPlus_V6;
   //    StoperReset_10 { ExternalAccessible := 'False'; ExternalVisible := 'False'; ExternalWritable := 'False'; S7_SetPoint := 'True'} : G7_StepPlus_V6;
   //    StoperRelease_10 { ExternalAccessible := 'False'; ExternalVisible := 'False'; ExternalWritable := 'False'; S7_SetPoint := 'True'} : G7_StepPlus_V6;
   //    WaitPalletArive_7 { ExternalAccessible := 'False'; ExternalVisible := 'False'; ExternalWritable := 'False'; S7_SetPoint := 'True'} : G7_StepPlus_V6;
   //    TimeDelay_7 { ExternalAccessible := 'False'; ExternalVisible := 'False'; ExternalWritable := 'False'; S7_SetPoint := 'True'} : G7_StepPlus_V6;
   //    AriveTimeDelay_11 { ExternalAccessible := 'False'; ExternalVisible := 'False'; ExternalWritable := 'False'; S7_SetPoint := 'True'} : G7_StepPlus_V6;
   //    StoperReset_11 { ExternalAccessible := 'False'; ExternalVisible := 'False'; ExternalWritable := 'False'; S7_SetPoint := 'True'} : G7_StepPlus_V6;
   //    StoperRelease_11 { ExternalAccessible := 'False'; ExternalVisible := 'False'; ExternalWritable := 'False'; S7_SetPoint := 'True'} : G7_StepPlus_V6;
   //    WaitPalletArive_8 { ExternalAccessible := 'False'; ExternalVisible := 'False'; ExternalWritable := 'False'; S7_SetPoint := 'True'} : G7_StepPlus_V6;
   //    TimeDelay_8 { ExternalAccessible := 'False'; ExternalVisible := 'False'; ExternalWritable := 'False'; S7_SetPoint := 'True'} : G7_StepPlus_V6;
   //    "CheckMachine Mode_6" { ExternalAccessible := 'False'; ExternalVisible := 'False'; ExternalWritable := 'False'; S7_SetPoint := 'True'} : G7_StepPlus_V6;
   //    "CheckMachine Mode_7" { ExternalAccessible := 'False'; ExternalVisible := 'False'; ExternalWritable := 'False'; S7_SetPoint := 'True'} : G7_StepPlus_V6;
   //    "CheckMachine Mode_8" { ExternalAccessible := 'False'; ExternalVisible := 'False'; ExternalWritable := 'False'; S7_SetPoint := 'True'} : G7_StepPlus_V6;
   //    WaitAllStoperReset { ExternalAccessible := 'False'; ExternalVisible := 'False'; ExternalWritable := 'False'; S7_SetPoint := 'True'} : G7_StepPlus_V6;
   //    Step182 { ExternalAccessible := 'False'; ExternalVisible := 'False'; ExternalWritable := 'False'; S7_SetPoint := 'True'} : G7_StepPlus_V6;
   //    WaitPalletArive_9 { ExternalAccessible := 'False'; ExternalVisible := 'False'; ExternalWritable := 'False'; S7_SetPoint := 'True'} : G7_StepPlus_V6;
   //    TimeDelay_9 { ExternalAccessible := 'False'; ExternalVisible := 'False'; ExternalWritable := 'False'; S7_SetPoint := 'True'} : G7_StepPlus_V6;
   //    CheckMachineMode { ExternalAccessible := 'False'; ExternalVisible := 'False'; ExternalWritable := 'False'; S7_SetPoint := 'True'} : G7_StepPlus_V6;
   //    UnloadStoper_1 { ExternalAccessible := 'False'; ExternalVisible := 'False'; ExternalWritable := 'False'; S7_SetPoint := 'True'} : G7_StepPlus_V6;
   //    UnloadStoper_2 { ExternalAccessible := 'False'; ExternalVisible := 'False'; ExternalWritable := 'False'; S7_SetPoint := 'True'} : G7_StepPlus_V6;
   //    UnloadStoper_3 { ExternalAccessible := 'False'; ExternalVisible := 'False'; ExternalWritable := 'False'; S7_SetPoint := 'True'} : G7_StepPlus_V6;
   //    "Process Finish_1" { ExternalAccessible := 'False'; ExternalVisible := 'False'; ExternalWritable := 'False'; S7_SetPoint := 'True'} : G7_StepPlus_V6;
   //    "Process Finish_2" { ExternalAccessible := 'False'; ExternalVisible := 'False'; ExternalWritable := 'False'; S7_SetPoint := 'True'} : G7_StepPlus_V6;
   //    "Process Finish_3" { ExternalAccessible := 'False'; ExternalVisible := 'False'; ExternalWritable := 'False'; S7_SetPoint := 'True'} : G7_StepPlus_V6;
   //    "Process Finish_4" { ExternalAccessible := 'False'; ExternalVisible := 'False'; ExternalWritable := 'False'; S7_SetPoint := 'True'} : G7_StepPlus_V6;
   //    "Process Finish_5" { ExternalAccessible := 'False'; ExternalVisible := 'False'; ExternalWritable := 'False'; S7_SetPoint := 'True'} : G7_StepPlus_V6;
   //    "Process Finish_6" { ExternalAccessible := 'False'; ExternalVisible := 'False'; ExternalWritable := 'False'; S7_SetPoint := 'True'} : G7_StepPlus_V6;
   //    "Process Finish_7" { ExternalAccessible := 'False'; ExternalVisible := 'False'; ExternalWritable := 'False'; S7_SetPoint := 'True'} : G7_StepPlus_V6;
   //    "Process Finish_8" { ExternalAccessible := 'False'; ExternalVisible := 'False'; ExternalWritable := 'False'; S7_SetPoint := 'True'} : G7_StepPlus_V6;
   //    "Process Finish_9" { ExternalAccessible := 'False'; ExternalVisible := 'False'; ExternalWritable := 'False'; S7_SetPoint := 'True'} : G7_StepPlus_V6;
   //    "Process Finish_10" { ExternalAccessible := 'False'; ExternalVisible := 'False'; ExternalWritable := 'False'; S7_SetPoint := 'True'} : G7_StepPlus_V6;
   //    "Process Finish_11" { ExternalAccessible := 'False'; ExternalVisible := 'False'; ExternalWritable := 'False'; S7_SetPoint := 'True'} : G7_StepPlus_V6;
   // END_VAR
BEGIN
END_DATA_BLOCK
